// TIA Portal V20 export
TYPE "LConSMC_typeFrictionMeasurement_V2"
// Ein-/Ausgänge der Reibkennlinienmessung / In-/Outputs of the friction measurement
// stored: Access Published
   STRUCT
      in { S7_SetPoint := 'True'} : "LConSMC_typeFrictionMeasurementV2In";   // Inputs of the FB FrictionMeasurementV2
      out { S7_SetPoint := 'True'} : "LConSMC_typeFrictionMeasurementV2Out";   // Outputs of the FB FrictionMeasurementV2
   END_STRUCT;
END_TYPE
